{attribute 'GeneratedUsingTerminal: IODEVICETYPE_ETHERCATPROT'}
{attribute addProperty BoxType "IODEVICETYPE_ETHERCATPROT"}
{attribute addProperty Id "Beckhoff_EQ1xxxBeckhoff_EQ1xxx_F7C2863978Beckhoff_EQ2xxxBeckhoff_EQ2xxx_CD55E279247Beckhoff_EQ3xxxBeckhoff_EQ3xxx_7E855133718SyncUnitsSyncUnits_99E584AF18InputsInputs_25A0042B160OutputsOutputs_2397A10E106InfoDataInfoData_E68C61CD28"}
{attribute addProperty CRC "3624530900"}
{attribute addProperty Size "1355"}
TYPE EtherCAT_Master_EQxxxx_D809F3D4 :
STRUCT
	{attribute addProperty Name "Beckhoff_EQ1xxx"}
	{attribute addProperty PreviousPort "EtherCAT_Master_EQxxxx : Master"}
	Beckhoff_EQ1xxx : Beckhoff_EQ1xxx_F7C28639;
	{attribute addProperty Name "Beckhoff_EQ2xxx"}
	{attribute addProperty PreviousPort "Beckhoff EQ1xxx : C"}
	Beckhoff_EQ2xxx : Beckhoff_EQ2xxx_CD55E279;
	{attribute addProperty Name "Beckhoff_EQ3xxx"}
	{attribute addProperty PreviousPort "Beckhoff EQ2xxx : C"}
	Beckhoff_EQ3xxx : Beckhoff_EQ3xxx_7E855133;
	{attribute addProperty Name "SyncUnits"}
	SyncUnits : SyncUnits_99E584AF;
	{attribute addProperty Name "Inputs"}
	Inputs : Inputs_25A0042B;
	{attribute addProperty Name "Outputs"}
	Outputs : Outputs_2397A10E;
	{attribute addProperty Name "InfoData"}
	InfoData : InfoData_E68C61CD;
END_STRUCT
END_TYPE

(* stored: Version 1.2.0.0, ProductVersion 3.1.4024.9
   DUT EtherCAT_Master_EQxxxx_D809F3D4: Id {3d18e313-91d4-4230-b721-d30cdbb5f542} *)
